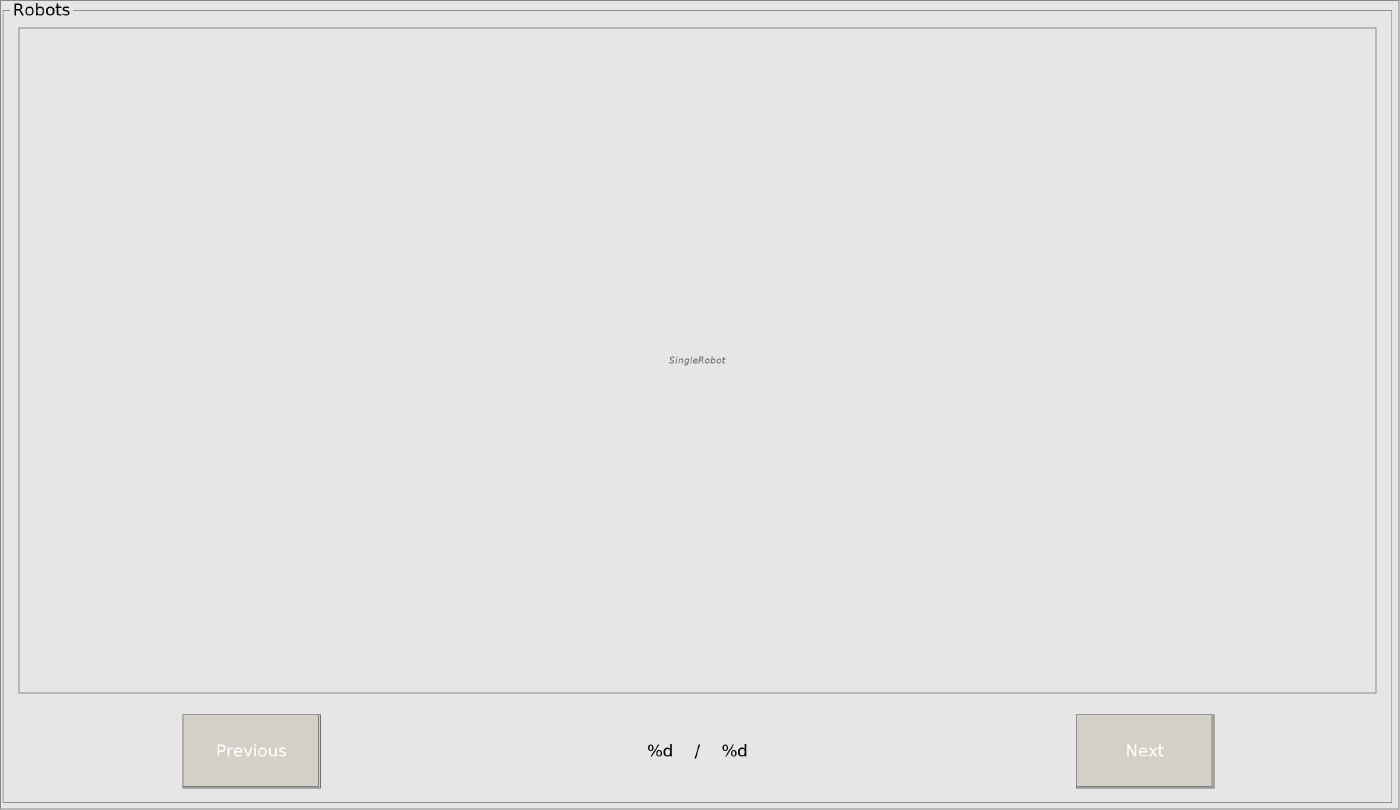
VISUALIZATION PageManualRobots_1  // 1520x880
VAR_IN_OUT
	btnPrevious			: BOOL;
	btnNext				: BOOL;
	bPreviousInvisible	: BOOL;
	bNextInvisible		: BOOL;
	stRobotEmpty		: ARRAY[1..1] OF BOOL;
	stRobot				: ARRAY[1..1] OF ST_VisuCtrlRobotFrame;
	iRobotSelectedPageIndex	: USINT;
	iRobotTotalPageIndex 	: USINT;
	
END_VAR
    GroupBox (3,3 1508x869), "Robots"
        Button (195,773 150x80), "Previous", invisible if: bPreviousInvisible
            tap btnPrevious
        Button (1165,773 150x80), "Next", invisible if: bNextInvisible
            tap btnNext
        Frame (17,27 1474x723), invisible if: stRobotEmpty[1]
            shows SingleRobot(stRobot := stRobot[1])
        Rectangle (689,788 130x50), "/"
        Rectangle (689,788 50x50), "%d", text variable: iRobotSelectedPageIndex+1
        Rectangle (770,788 50x50), "%d", text variable: iRobotTotalPageIndex+1
END_VISUALIZATION

(* stored: Version 1.1.0.1, ProductVersion 3.1.4024.12
   Visu PageManualRobots_1: Id {8961480b-6656-4b13-a6d7-6d66155b1fa7} *)
